Staubli VAL3: oPilatusCover.pgx

public program oPilatusCover(num nChoice (dimensions=1))
// oPilatusCover
begin
  dioSet(oPilatusCover,nChoice)
end
